//{attribute 'qualified_only'}
VAR_GLOBAL
	//
END_VAR

VAR_GLOBAL
	//g_slaveInfo:ARRAY[1..g_sJntNum] OF ST_JntInfo;
	//g_SetupInfo:ARRAY[1..g_setupJntNum] OF ST_JntInfo;
	//g_cartInfo:ARRAY[1..g_sJntNum] OF ST_JntInfo;
END_VAR

(* stored: Version 1.1.0.1, ProductVersion 3.1.4024.11
   GVL GVL_Define: Id {3910f9b4-7711-46b6-8904-bcd582bf4526} *)
